// TIA Portal V17 export
// export: Created 2023-12-22T15:03:16.1136124Z, ExportSetting WithDefaults, DisplayName Totally Integrated Automation Portal, DisplayVersion V17, DisplayName TIA Portal Openness, DisplayVersion V17, DisplayName TIA Portal Version Control Interface, DisplayVersion V17, DisplayName STEP 7 Professional, DisplayVersion V17, DisplayName STEP 7 Safety, DisplayVersion V17, DisplayName WinCC Advanced, DisplayVersion V17
DATA_BLOCK "Comm_SKV_14"   // DB1014
VERSION : 0.1
// stored: AutoNumber false, DBAccessibleFromOPCUA true, DBAccessibleFromWebserver true, InstanceOfName Comm_SKV, InstanceOfType FB
"Comm_SKV"
   // VAR RETAIN
   //    To_SKV : Struct
   //       watchdog : Int;
   //       LE_1 : Int;
   //       LE_2 : Int;
   //       LE_3 : Int;
   //       LE_4 : Int;
   //       SP_FE : Int;
   //       SP_M : Int;
   //       CMD : Struct
   //          REQ : Bool;
   //          Reset : Bool;
   //          Hand : Bool;
   //          Start_M : Bool;
   //       END_STRUCT;
   //       Valves : Struct
   //          ID : Int;
   //          Local : Array[0..15] of Bool;
   //          Mode : Array[1..10] of Int;
   //          Status : Array[1..10] of Int;
   //       END_STRUCT;
   //    END_STRUCT;
   //    From_SKV : Struct
   //       watchdog : Int;
   //       LE_SKV : Int;
   //       res_h : DInt;
   //       LE : Int;
   //       TE : Int;
   //       PE_1 : Int;
   //       PE_2 : Int;
   //       PE_3 : Int;
   //       PE_4 : Int;
   //       FE : Int;
   //       C : Int;
   //       Status : Int;
   //       STATE : Struct
   //          Ready : Bool;
   //          Local : Bool;
   //          Warning : Bool;
   //          Alarm : Bool;
   //          LS : Bool;
   //          Lock : Bool;
   //       END_STRUCT;
   //       Valves : Struct
   //          ID : Int;
   //          REQ : Array[0..15] of Bool;
   //       END_STRUCT;
   //    END_STRUCT;
   //    watchdog_control : Int;
   //    Alarm : Struct
   //       Link : Bool;
   //    END_STRUCT;
   //    ID : Int;
   //    SP_M : Real;
   //    SP_FE : Real;
   //    LE : Real;
   //    PE_1 : Real;
   //    PE_2 : Real;
   //    PE_3 : Real;
   //    PE_4 : Real;
   //    FE : Real;
   //    TE : Real;
   //    C : Real;
   //    Route : Bool;
   //    "Name" : Array[0..10] of String[5];
   //    Clock : Array[0..10] of "Time_S";
   // END_VAR
BEGIN
END_DATA_BLOCK
